// TIA Portal V20 export
TYPE "LER_typeStatusCamIn"
// stored: Access Published
   STRUCT
      InSync : Bool;
      Busy : Bool;
      Error : Bool;
      ErrorId : Word;
   END_STRUCT;
END_TYPE
